// TIA Portal V20 export
TYPE "typePhmi"
// stored: Access Published, IsFailsafeCompliant true, Namespace Safety
   STRUCT
      estop : Bool;   // Emergency Button
      enable : Bool;   // DeadMan Switch
      reset : Bool;
      PhmiForcedDisconnection : Bool;   // Phmi Forced Disconnection
   END_STRUCT;
END_TYPE
